// TIA Portal V16 export
// export: Created 2021-07-12T14:47:20.7397065Z, ExportSetting WithDefaults, DisplayName Totally Integrated Automation Portal, DisplayVersion V16, DisplayName TIA Portal Version Control Interface, DisplayVersion V16, DisplayName TIA Portal Openness, DisplayVersion V16, DisplayName STEP 7 Professional, DisplayVersion V16, DisplayName STEP 7 Safety, DisplayVersion V16, DisplayName WinCC Professional, DisplayVersion V16
TYPE "SimaHydTO_typeHMIConnectionAxisToDataErrorDetail"
TITLE = SimaHydTO_typeHMIConnectionAxisToDataErrorDetail
// HMI interface: Technology object axis error detail
// stored: IsFailsafeCompliant false
   STRUCT
      number : UDInt;   // Error number
      reaction : DInt;   // Error reaction
   END_STRUCT;
END_TYPE
